(* PLC project M3_16, Desconocido M3_16 1 *)
(* stored: creationDateTime 2025-05-15T11:40:54, modificationDateTime 2025-05-15T14:50:20 *)

PROGRAM Main
  VAR
    CTU0 : CTU;
    xPulso : BOOL;
    xReset : BOOL;
    xConteoFinalizado : BOOL;
    iConteo : INT;
  END_VAR
  VAR  (* added by the conversion: wires and edge detectors of the diagram *)
    R_TRIG1 : R_TRIG;
  END_VAR

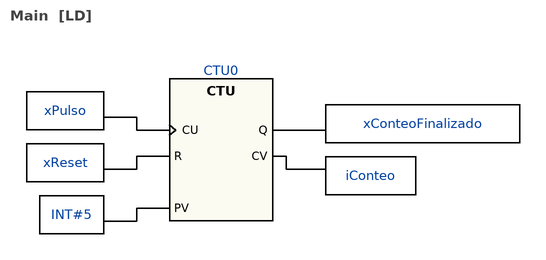
(* LD diagram, written out as Structured Text *)
R_TRIG1(CLK := xPulso);
CTU0(CU := R_TRIG1.Q, R := xReset, PV := INT#5);
iConteo := CTU0.CV;
xConteoFinalizado := CTU0.Q;
END_PROGRAM

CONFIGURATION Config0
  RESOURCE Res0 ON PLC
    TASK task0(INTERVAL := T#20ms, PRIORITY := 0);
    PROGRAM instance0 WITH task0 : Main;
  END_RESOURCE
END_CONFIGURATION
